// TIA Portal V16 export
// export: Created 2024-08-24T20:10:16.4979602Z, ExportSetting WithDefaults, DisplayName Totally Integrated Automation Portal, DisplayVersion V16, DisplayName TIA Portal Version Control Interface, DisplayVersion V16, DisplayName TIA Portal Openness, DisplayVersion V16, DisplayName STEP 7 Professional, DisplayVersion V16, DisplayName STEP 7 Safety, DisplayVersion V16, DisplayName WinCC Professional, DisplayVersion V16
VAR_GLOBAL   // PLC tag table "Tabla de variables estándar"
   Tag_1 AT %M10.0 : Bool;
   Tag_2 AT %M10.1 : Bool;
   Tag_3 AT %M10.2 : Bool;
   Tag_4 AT %M10.3 : Bool;
END_VAR
